{attribute 'qualified_only'}
VAR_GLOBAL
END_VAR

(* stored: Version 1.1.0.1, ProductVersion 3.1.4024.13
   GVL GVL: Id {50f19d3f-afc1-43c5-b2e3-aa11f6342f97} *)
